(* PLC project Senza_nome, Sconosciuto Senza_nome 1 *)
(* stored: creationDateTime 2020-05-23T16:03:02, modificationDateTime 2020-05-27T15:09:30 *)

PROGRAM manageLights
  VAR_EXTERNAL
    startButton : BOOL;
    stopButton : BOOL;
    startLight : BOOL;
    stopLight : BOOL;
    fillValveMan : BOOL;
    dischargeValveMan : BOOL;
    fillManualLight : BOOL;
    dischargeManualLight : BOOL;
    manual : BOOL;
  END_VAR
  VAR
    aux1 : BOOL;
    aux2 : BOOL;
  END_VAR
  VAR  (* added by the conversion: wires and edge detectors of the diagram *)
    R_TRIG1 : R_TRIG;
    R_TRIG2 : R_TRIG;
    F_TRIG3 : F_TRIG;
    R_TRIG4 : R_TRIG;
  END_VAR

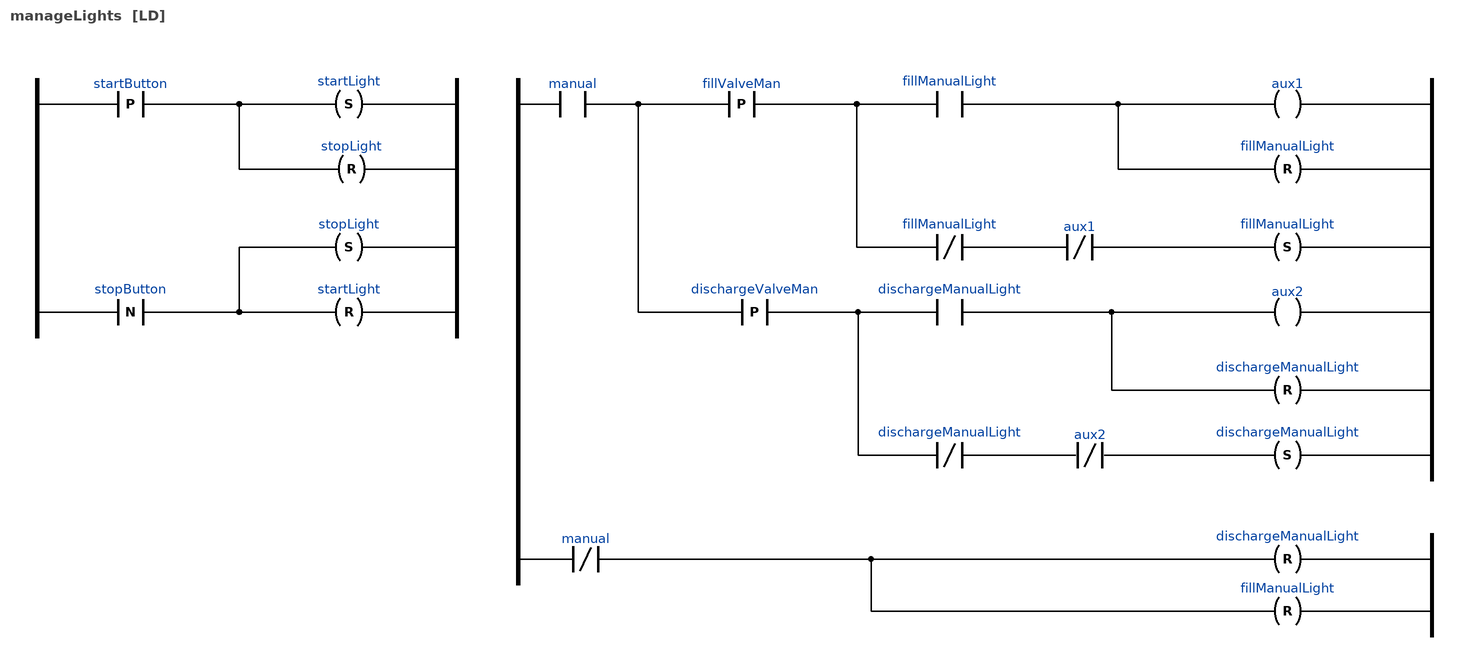
(* LD diagram, written out as Structured Text *)
R_TRIG1(CLK := startButton);
IF R_TRIG1.Q THEN startLight := TRUE; END_IF;
R_TRIG2(CLK := fillValveMan);
aux1 := manual AND R_TRIG2.Q AND fillManualLight;
IF R_TRIG1.Q THEN stopLight := FALSE; END_IF;
IF manual AND R_TRIG2.Q AND fillManualLight THEN fillManualLight := FALSE; END_IF;
F_TRIG3(CLK := stopButton);
IF F_TRIG3.Q THEN stopLight := TRUE; END_IF;
IF manual AND R_TRIG2.Q AND NOT fillManualLight AND NOT aux1 THEN fillManualLight := TRUE; END_IF;
IF F_TRIG3.Q THEN startLight := FALSE; END_IF;
R_TRIG4(CLK := dischargeValveMan);
aux2 := manual AND R_TRIG4.Q AND dischargeManualLight;
IF manual AND R_TRIG4.Q AND dischargeManualLight THEN dischargeManualLight := FALSE; END_IF;
IF manual AND R_TRIG4.Q AND NOT dischargeManualLight AND NOT aux2 THEN dischargeManualLight := TRUE; END_IF;
IF NOT manual THEN dischargeManualLight := FALSE; END_IF;
IF NOT manual THEN fillManualLight := FALSE; END_IF;
END_PROGRAM

(* Gestione display *)
PROGRAM manageDisplays
  VAR_EXTERNAL
    levelMeter : INT;
    flowMeter : INT;
    setpoint : INT;
    Kp : INT;
    Ki : INT;
    Kd : INT;
    dischargeValve : INT;
    dischargeValvePos : INT;
    fillValve : INT;
    fillValvePos : INT;
    KpVal : INT;
    KiVal : INT;
    KdVal : INT;
    setpointVal : INT;
    errorVal : INT;
    levelVal : INT;
  END_VAR
  VAR
    levelConvFactor : REAL := 3.34;  (* Conversion factor from level meter to actual scale *)
    setpointConvFactor : REAL := 3.34;  (* Conversion factor from potentiometer (0-1000) to setpoint (0-300) *)
    KpConvFactor : INT := 10;  (* Conversion factor for PID gains *)
    KiConvFactor : INT := 10;  (* Conversion factor for PID gains *)
    KdConvFactor : INT := 10;  (* Conversion factor for PID gains *)
  END_VAR

            dischargeValvePos := dischargeValve;
fillValvePos := fillValve;
KpVal := Kp/KpConvFactor;
KiVal := Ki/KiConvFactor;
KdVal := Kd/KdConvFactor;
setpointVal := REAL_TO_INT(DIV(INT_TO_REAL(setpoint), setpointConvFactor));
levelVal := REAL_TO_INT(DIV(INT_TO_REAL(levelMeter), levelConvFactor));
errorVal := setpointVal - levelVal;

          
END_PROGRAM

PROGRAM manualMode
  VAR_EXTERNAL
    manual : BOOL;
    startLight : BOOL;
    stopLight : BOOL;
    fillManualLight : BOOL;
    dischargeManualLight : BOOL;
    fillValve : INT;
    dischargeValve : INT;
  END_VAR

            IF manual&startLight THEN
  IF fillManualLight THEN
    fillValve := 10*100;
  ELSE
    fillValve := 0; 
  END_IF;
  
  IF dischargeManualLight THEN
    dischargeValve := 10*100;
  ELSE
    dischargeValve := 0; 
  END_IF;

ELSIF manual&stopLight THEN
  fillValve := 0;
  dischargeValve := 0;
END_IF;
          
END_PROGRAM

PROGRAM autoMode
  VAR_EXTERNAL
    auto : BOOL;
    startLight : BOOL;
    setpointVal : INT;
    levelVal : INT;
    fillValve : INT;
    dischargeValve : INT;
    KpVal : INT;
    KiVal : INT;
    KdVal : INT;
  END_VAR
  VAR
    Kp_internal : REAL;
    Ki_internal : REAL;
    Kd_internal : REAL;
    Ti_internal : REAL;
    Td_internal : REAL;
    setpoint_internal : REAL;
    level_internal : REAL;
    cycle : TIME := T#20ms;
    PID_level : PID;
    control : REAL;
    Kpmax : REAL := 100.0;
    Kimax : REAL := 0.1;
    Kdmax : REAL := 10.0;
    pippo : PID;
  END_VAR

            Kp_internal := INT_TO_REAL(KpVal)/100.0*Kpmax;
Ki_internal := INT_TO_REAL(KiVal)/100.0*Kimax;
Kd_internal := INT_TO_REAL(KdVal)/100.0*Kdmax;

setpoint_internal := INT_TO_REAL(setpointVal);
level_internal := INT_TO_REAL(levelVal);

IF GT(Ki_internal,0.0) THEN
  Ti_internal := Kp_internal/Ki_internal;
ELSE
  Ti_internal := 100000000000000000.0; (* just a very big number to put Ki \approx. 0 *)
END_IF;

IF (GT(Kd_internal,0.0)&NE(Kp_internal,0.0)) THEN
  Td_internal := Kd_internal/Kp_internal;
ELSE
  Td_internal := 0.0;
END_IF;

PID_level(
     AUTO := auto,
     PV := level_internal, (* process variable *)
     SP := setpoint_internal,
     X0 := 0.0, (* default when auto=false *)
     KP := Kp_internal,
     TR := Ti_internal,
     TD := Td_internal,
     CYCLE := cycle,
     XOUT => control);

control := -control; (* OpenPLC does PV-SP *)
IF auto&startLight THEN
  IF GT(control, 0.0) THEN
    fillValve := REAL_TO_INT(control);
    dischargeValve := 0;
  ELSE
    fillValve := 0;
    dischargeValve := REAL_TO_INT(-control);
  END_IF;

END_IF;

          
END_PROGRAM

CONFIGURATION Config0
  RESOURCE Res0 ON PLC
    VAR_GLOBAL
      startButton AT %IX100.0 : BOOL;
      stopButton AT %IX100.1 : BOOL;
      manual AT %IX100.2 : BOOL;
      auto AT %IX100.3 : BOOL;
      fillValveMan AT %IX100.4 : BOOL;
      dischargeValveMan AT %IX100.5 : BOOL;
      startLight AT %QX100.0 : BOOL;
      stopLight AT %QX100.1 : BOOL;
      fillManualLight AT %QX100.2 : BOOL;
      dischargeManualLight AT %QX100.3 : BOOL;
      levelMeter AT %IW100 : INT;
      flowMeter AT %IW101 : INT;
      setpoint AT %IW102 : INT;
      Kp AT %IW103 : INT;
      Ki AT %IW104 : INT;
      Kd AT %IW105 : INT;
      dischargeValve AT %QW100 : INT;
      dischargeValvePos AT %QW101 : INT;
      fillValve AT %QW102 : INT;
      fillValvePos AT %QW103 : INT;
      KpVal AT %QW104 : INT;
      KiVal AT %QW105 : INT;
      KdVal AT %QW106 : INT;
      setpointVal AT %QW107 : INT;
      errorVal AT %QW108 : INT;
      levelVal AT %QW109 : INT;
    END_VAR
    TASK task0(INTERVAL := T#20ms, PRIORITY := 0);
    TASK task1(INTERVAL := T#200ms, PRIORITY := 2);
    PROGRAM instance1 WITH task0 : manageDisplays;
    PROGRAM instance2 WITH task0 : manualMode;
    PROGRAM instance3 WITH task0 : autoMode;
    PROGRAM instance0 WITH task1 : manageLights;
  END_RESOURCE
END_CONFIGURATION
